// TwinCAT 3 PLC project MES_Lib
// Title: VM MES
// Company: Vesz-Mont 2000 KFT.
// Author: Zsolt Závori
// ProjectVersion: 1.0.0
// ProgramVersion: 3.1.4023.0
// libraries:
//   Tc2_Standard, * (Beckhoff Automation GmbH)
//   Tc2_System, * (Beckhoff Automation GmbH)
//   Tc2_TcpIp, * (Beckhoff Automation GmbH)
//   Tc2_Utilities, * (Beckhoff Automation GmbH)
//   Tc3_IotBase, * (Beckhoff Automation GmbH)
//   Tc3_JsonXml, * (Beckhoff Automation GmbH)
//   Tc3_Module, * (Beckhoff Automation GmbH)
// project tree:
//   DUTs/ I_SR1000.TcIO, ST_Field.TcDUT
//   FBs/ FB_GET_Base.TcPOU, FB_NextPhase.TcPOU, FB_TCP_IP.TcPOU
//   GVLs/ ComPar.TcGVL
//   / PlcTask.TcTTO
//   Test/ Test.TcPOU
// real-time tasks:
//   TASK PlcTask: cycle T#10ms, priority 20, ADS port 350

CONFIGURATION MES_Lib
    RESOURCE PLC ON TwinCAT3
        TASK PlcTask(INTERVAL := T#10ms, PRIORITY := 20);
        PROGRAM Test WITH PlcTask : Test;
    END_RESOURCE
END_CONFIGURATION

// ---- DUTs/ST_Field.TcDUT
TYPE ST_Field :
STRUCT
	FieldName			: STRING(255);
	FieldValue			: STRING(255);
END_STRUCT
END_TYPE

// ---- GVLs/ComPar.TcGVL
{attribute 'qualified_only'}
VAR_GLOBAL
	HostName				: STRING := '192.168.216.149';
	HostPort				: UINT := 19000;
END_VAR

// ---- DUTs/I_SR1000.TcIO
INTERFACE I_SR1000

END_INTERFACE

// ---- Test/Test.TcPOU
PROGRAM Test
VAR
	fbSR1000						:FB_TCP_IP;
	sCode							:STRING;
	nErrorId						:UDINT;
	bTrigger						:BOOL;

	fbCloseAll						:FB_SocketCloseAll;
	bInitTCPIP						:BOOL;
	bInit							:BOOL := TRUE;
	
	stFields						: ARRAY [0..1] OF ST_Field := [ (FieldName := 'x-api-key', FieldValue := '5308cb47-0343-498d-a4d9-dac5c6a15f1e'), 
																	(FieldName := 'x-terminal-token', FieldValue := 'logistic')];
	fbNextPhase						: FB_NextPhase;
											
END_VAR

IF bInit THEN
	Init();
END_IF


fbCloseAll( sSrvNetID := '', bExecute:= bInitTCPIP );
IF NOT fbCloseAll.bBusy AND bInitTCPIP THEN
	bInitTCPIP := FALSE;
END_IF



IF bTrigger THEN
	IF fbSR1000.ReadSR1000(sCode, nErrorId) THEN
		bTrigger := FALSE;
	END_IF
END_IF

fbNextPhase(stFields := stFields);
fbNextPhase.GET();

ACTION Init:
	fbSR1000.p_ConnectTimeout := T#2S;
	fbSR1000.p_SendTimeout := T#2S;
	fbSR1000.p_ReceiveTimeout := T#2S;
	fbSR1000.p_CloseTimeout := T#2S;
	fbSR1000(sName:= 'SR1000', sRemoteHost:= '192.168.216.96', nRemotePort:= 9004);
	bInit := FALSE;
END_ACTION

END_PROGRAM

// ---- FBs/FB_TCP_IP.TcPOU
FUNCTION_BLOCK FB_TCP_IP
VAR_INPUT
	sName				: STRING := 'SR1000';			(* A kódolvasó neve *)
	sRemoteHost			: STRING(15) := '127.0.0.1';	(* IP adress of remote server *)
	nRemotePort			: UDINT := 9004;				(* SR1000 default port *)
END_VAR
VAR_OUTPUT
END_VAR
VAR
	fbConnect 			:FB_SocketConnect;
	fbSend 				:FB_SocketSend;
	fbReceive 			:FB_SocketReceive;
	fbClose				:FB_SocketClose;
	sTxBuffer			:STRING;
	sRxBuffer			:STRING;
	nStep				:INT := 0;
	
	_ConnectTimeout		:TIME;
	_SendTimeout		:TIME;
	_ReceiveTimeout		:TIME;
	_CloseTimeout		:TIME;

END_VAR

(*
fbConnect(
	sSrvNetId:= '', 
	sRemoteHost:= sRemoteHost, 
	nRemotePort:= nRemotePort, 
	bExecute:= , 
	tTimeout:= _ConnectTimeout, 
	bBusy=> , 
	bError=> , 
	nErrId=> , 
	hSocket=> );
	
fbSend(
	sSrvNetId:= '', 
	hSocket:= fbConnect.hSocket, 
	cbLen:= INT_TO_UDINT(LEN(sTxBuffer)), 
	pSrc:= ADR(sTxBuffer), 
	bExecute:= , 
	tTimeout:= _SendTimeout, 
	bBusy=> , 
	bError=> , 
	nErrId=> );

fbReceive(
	sSrvNetId:= '', 
	hSocket:= fbConnect.hSocket, 
	cbLen:= SIZEOF(sRxBuffer), 
	pDest:= ADR(sRxBuffer), 
	bExecute:= , 
	tTimeout:= _ReceiveTimeout, 
	bBusy=> , 
	bError=> , 
	nErrId=> , 
	nRecBytes=> );

fbClose(
	sSrvNetId:= '', 
	hSocket:= fbConnect.hSocket, 
	bExecute:= , 
	tTimeout:= , 
	bBusy=> , 
	bError=> , 
	nErrId=> );	
	
*)

PROPERTY p_CloseTimeout :  TIME
GET
p_CloseTimeout := _CloseTimeout;
END_GET
SET
IF p_CloseTimeout > T#100MS AND p_CloseTimeout <  T#60S THEN
	_CloseTimeout := p_CloseTimeout;
ELSE
	_CloseTimeout := T#1S;					// default value
END_IF
END_SET
END_PROPERTY

PROPERTY p_ConnectTimeout : TIME
GET
p_ConnectTimeout := _ConnectTimeout;
END_GET
SET
IF p_ConnectTimeout > T#100MS AND p_ConnectTimeout <  T#60S THEN
	_ConnectTimeout := p_ConnectTimeout;
ELSE
	_ConnectTimeout := T#1S;					// default value
END_IF
END_SET
END_PROPERTY

PROPERTY p_ReceiveTimeout : TIME
GET
p_ReceiveTimeout := _ReceiveTimeout;
END_GET
SET
IF p_ReceiveTimeout > T#100MS AND p_ReceiveTimeout <  T#60S THEN
	_ReceiveTimeout := p_ReceiveTimeout;
ELSE
	_ReceiveTimeout := T#1S;					// default value
END_IF
END_SET
END_PROPERTY

PROPERTY p_SendTimeout : TIME
GET
p_SendTimeout := _SendTimeout;
END_GET
SET
IF p_SendTimeout > T#100MS AND p_SendTimeout <  T#60S THEN
	_SendTimeout := p_SendTimeout;
ELSE
	_SendTimeout := T#1S;					// default value
END_IF
END_SET
END_PROPERTY

METHOD ReadSR1000 : BOOL
VAR_INPUT
	sCode						:REFERENCE TO STRING;
	nErrorId					:REFERENCE TO UDINT;
END_VAR
TCP_Com();
ReadSR1000 := FALSE;
CASE nStep OF
0:		fbConnect.bExecute := TRUE;
		sRxBuffer := '';
		nStep := nStep + 20;
	
20:		IF NOT fbConnect.bBusy THEN
			fbConnect.bExecute := FALSE;
			nStep := nStep + 20;
		ELSIF fbConnect.bError THEN
			sCode := '';
			nErrorId := fbConnect.nErrId;
			fbConnect.bExecute := FALSE;
			nStep := 200;
		END_IF
	
40:		sTxBuffer := 'LON$R$N';
		fbSend.bExecute := TRUE;
		nStep := nStep + 20;
	
60:		IF NOT fbSend.bBusy THEN
			fbSend.bExecute := FALSE;
			nStep := 100;
		ELSIF fbSend.bError THEN
			sCode := '';
			nErrorId := fbSend.nErrId;
			fbSend.bExecute := FALSE;
			nStep := 200;
		END_IF
	
100:	fbReceive.bExecute := TRUE;
		nStep := nStep + 20;
	
120:	IF NOT fbReceive.bBusy THEN
			IF NOT fbReceive.bError THEN
					fbReceive.bExecute := FALSE;
					nStep := nStep + 20;
			ELSE
					sCode := '';
					nErrorId := fbReceive.nErrId;
					fbReceive.bExecute := FALSE;
					nStep := 200;
			END_IF
		END_IF

140:	IF fbReceive.nRecBytes > 0 THEN
				IF MID(sRxBuffer, 1, UDINT_TO_INT(fbReceive.nRecBytes)) = '$0D' THEN
					nErrorId := fbReceive.nErrId;
					sCode := LEFT(sRxBuffer, UDINT_TO_INT(fbReceive.nRecBytes)-1);
					nStep := 200;
				ELSE				
					nStep := 100;
				END_IF
		ELSE
				nStep := 100;
		END_IF
		
200:	fbClose.bExecute := TRUE;
		nStep := nStep + 20;
	
220:	IF NOT fbClose.bBusy THEN
			fbClose.bExecute := FALSE;
			nStep := 500;
		ELSIF fbClose.bError THEN
			sCode := '';
			nErrorId := fbClose.nErrId;
			fbClose.bExecute := FALSE;
			nStep := 500;
		END_IF

500:
		ReadSR1000 := TRUE;
		nStep := 0;
END_CASE
END_METHOD

METHOD PRIVATE TCP_Com : BOOL
VAR_INPUT
END_VAR
fbConnect(
	sSrvNetId:= '', 
	sRemoteHost:= sRemoteHost, 
	nRemotePort:= nRemotePort, 
	bExecute:= , 
	tTimeout:= _ConnectTimeout, 
	bBusy=> , 
	bError=> , 
	nErrId=> , 
	hSocket=> );
	
fbSend(
	sSrvNetId:= '', 
	hSocket:= fbConnect.hSocket, 
	cbLen:= INT_TO_UDINT(LEN(sTxBuffer)), 
	pSrc:= ADR(sTxBuffer), 
	bExecute:= , 
	tTimeout:= _SendTimeout, 
	bBusy=> , 
	bError=> , 
	nErrId=> );

fbReceive(
	sSrvNetId:= '', 
	hSocket:= fbConnect.hSocket, 
	cbLen:= SIZEOF(sRxBuffer), 
	pDest:= ADR(sRxBuffer), 
	bExecute:= , 
	tTimeout:= _ReceiveTimeout, 
	bBusy=> , 
	bError=> , 
	nErrId=> , 
	nRecBytes=> );

fbClose(
	sSrvNetId:= '', 
	hSocket:= fbConnect.hSocket, 
	bExecute:= , 
	tTimeout:= , 
	bBusy=> , 
	bError=> , 
	nErrId=> );
END_METHOD

END_FUNCTION_BLOCK

// ---- FBs/FB_NextPhase.TcPOU
FUNCTION_BLOCK FB_NextPhase
VAR_INPUT
	bSend							: BOOL;
	sSerialNr						: STRING;
END_VAR
VAR_IN_OUT
	stFields						: ARRAY [*] OF ST_Field;
END_VAR
VAR_OUTPUT
	bBusy							: BOOL;
	bError							: BOOL;
	sNextPhase						: STRING;
END_VAR
VAR
	fbJson     						: FB_JsonDomParser;
	jsonDoc							: SJsonValue;
	jsonBegin						: SJsonValue;
	jsonElement						: SJsonValue;
	jsonValue						: SJsonValue;
	fbGetWorkpieceData				: FB_GET_Base;
	nWorkPieceId					: ULINT;
	fbGetNextPhase					: FB_GET_Base;
	nState							: UDINT;
	RisingEdge						: R_TRIG;
	
END_VAR

fbGetWorkpieceData(sUri:= CONCAT('/api/workpieces/?serialNumber=', sSerialNr), stFields := stFields);
fbGetWorkpieceData.GET();

fbGetNextPhase(sUri:= CONCAT(CONCAT('/api/workpieces/', ULINT_TO_STRING(nWorkPieceId)), '/next-phases-resources'), stFields := stFields);
fbGetNextPhase.GET();

METHOD GET : BOOL
VAR_INPUT
END_VAR
RisingEdge(CLK:= bSend );
CASE nState OF
0:	
	IF RisingEdge.Q THEN
		fbGetWorkpieceData.bSend := TRUE; 						
		nState := nState +20;
		bBusy:= TRUE;
		bError:= FALSE;
	END_IF
	
20:
	IF NOT fbGetWorkpieceData.bBusy THEN
		fbGetWorkpieceData.bSend := FALSE;
		jsonDoc := fbJson.ParseDocument(fbGetWorkpieceData.sResult);
		jsonElement := fbJson.GetArrayValueByIdx(jsonDoc, 0);
		jsonValue := fbJson.FindMember(jsonElement, 'id');
		nWorkPieceId := LINT_TO_ULINT(fbJson.GetInt64(jsonValue));
		nState := nState +20; 
	END_IF
	
40:	
	fbGetNextPhase.bSend := TRUE;
	nState := nState +20;
	
60:
	IF NOT fbGetNextPhase.bBusy THEN
		fbGetNextPhase.bSend := FALSE;
		jsonDoc := fbJson.ParseDocument(fbGetNextPhase.sResult);
		jsonElement := fbJson.FindMember(jsonDoc, 'phase');
		jsonValue := fbJson.FindMember(jsonElement, 'name');
		sNextPhase := fbJson.GetString(jsonValue);
		nState := 0;
		bBusy:= FALSE;
	END_IF
END_CASE
END_METHOD

END_FUNCTION_BLOCK

// ---- FBs/FB_GET_Base.TcPOU
FUNCTION_BLOCK FB_GET_Base
VAR_INPUT
	bSend				: BOOL;
	sUri				: STRING;
END_VAR
VAR_IN_OUT
	stFields			: ARRAY [*] OF ST_Field;
END_VAR
VAR_OUTPUT
	bBusy				: BOOL;
	bError				: BOOL;
END_VAR
VAR
	fbClient			: FB_IotHttpClient;
	fbRequest			: FB_IotHttpRequest;
	fbHeader			: FB_IotHttpHeaderFieldMap;
	fbJson				: FB_JsonDomParser;
	nState				: UDINT;
	RisingEdge			: R_TRIG;
	
	bGetContentResult	: BOOL;
	sContent			: STRING(2000);
	
	bGetJsonResult		: BOOL;
	sResult				: STRING(2000);
	
	nReqCount			: UDINT;	
	nResCount			: UDINT;
	nValidResCount		: UDINT;
	nErrCount			: UDINT;
	bOnce				: BOOL:= TRUE;
	i					: DINT;
END_VAR

IF bOnce THEN
	FOR i := LOWER_BOUND(stFields,1) TO UPPER_BOUND(stFields,1) DO
		fbHeader.AddField(stFields[i].FieldName,stFields[i].FieldValue,FALSE);
	END_FOR	
	bOnce:= FALSE;
END_IF

IF NOT fbClient.bConfigured THEN
 	fbClient.sHostName := ComPar.HostName;
	fbClient.nHostPort:= ComPar.HostPort;
	fbClient.bKeepAlive := TRUE;
	fbClient.tConnectionTimeout := T#10s;
END_IF

fbClient.Execute();

METHOD GET : BOOL
VAR_INPUT
END_VAR
RisingEdge(CLK:= bSend );
CASE nState OF
0:	
	IF RisingEdge.Q THEN 
		IF fbRequest.SendRequest(sUri:= sUri, fbClient:=fbClient, eRequestType:=ETcIotHttpRequestType.HTTP_Get, 0, 0, fbHeader) THEN				
			nState:= 1;
			nReqCount:= nReqCount+1;
			bBusy:= TRUE;
			bError:= FALSE;
		END_IF					
	END_IF
1:
	IF NOT fbRequest.bBusy THEN
		bError:= TRUE;
		IF NOT fbRequest.bError THEN				 
			bGetContentResult:= fbRequest.GetContent(pContent:= ADR(sContent), nContentSize:= SIZEOF(sContent), bSetNullTermination:= TRUE);
			IF fbRequest.nStatusCode >= 200 AND fbRequest.nStatusCode < 300 THEN
				bGetJsonResult:= FALSE;
				IF fbRequest.GetJsonDomContent(fbJson) <> 0 THEN
					bGetJsonResult:= TRUE;
					nValidResCount:= nValidResCount+1;
					UTF8_TO_STRING(ADR(sResult),ADR(sContent),SIZEOF(sResult));
					bError:= FALSE;															
				END_IF							
				nResCount:= nResCount+1;			
			END_IF
		END_IF
		nState:= 0;
		GET := TRUE;
		bBusy:= FALSE;
		IF bError THEN
			nErrCount:= nErrCount+1;
		END_IF
	END_IF

END_CASE
END_METHOD

END_FUNCTION_BLOCK
